Staubli VAL3: iLevelFault.pgx

public program iLevelFault(num& nNum[] (dimensions=1))
begin
  nNum=dioGet(iLevelFault)
end
